# EPICS alarm handler configuration: mps_database/bareTest/alarms/areas/mpln_col0_mp01.alhConfig
GROUP NULL MPLN:COL0:MP01:1
$ALIAS MPS Link Node 56
$GUIDANCE
LTUH MPS
   Group Name: MPLN:COL0:MP01:1
   Summary PV:  MPLN:COL0:MP01:1:STATSUMY
$END
CHANNEL  MPLN:COL0:MP01:1    MPLN:COL0:MP01:1:MPS_EN_RBV		-----
CHANNEL  MPLN:COL0:MP01:1    MPLN:COL0:MP01:1:LC1_MODE_RBV		-----
